// TIA Portal V20 export
FUNCTION_BLOCK "F-FB_DigitalOutput"   // FB111, F_LAD
{ S7_Optimized_Access := 'TRUE' }
// stored: AutoNumber false
BEGIN

REGION Network 1: Contactor for Machine
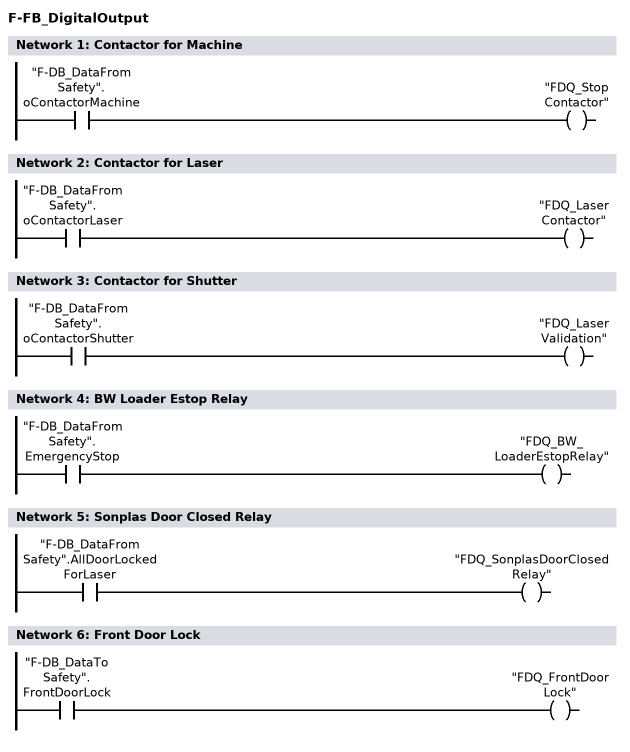
   RUNG wire#powerrail
      Contact( "F-DB_DataFromSafety".oContactorMachine )
      Coil( "FDQ_StopContactor" )
   END_RUNG
   // the same network as SCL:
   "FDQ_StopContactor" := "F-DB_DataFromSafety".oContactorMachine;
END_REGION

REGION Network 2: Contactor for Laser
   RUNG wire#powerrail
      Contact( "F-DB_DataFromSafety".oContactorLaser )
      Coil( "FDQ_LaserContactor" )
   END_RUNG
   // the same network as SCL:
   "FDQ_LaserContactor" := "F-DB_DataFromSafety".oContactorLaser;
END_REGION

REGION Network 3: Contactor for Shutter
   RUNG wire#powerrail
      Contact( "F-DB_DataFromSafety".oContactorShutter )
      Coil( "FDQ_LaserValidation" )
   END_RUNG
   // the same network as SCL:
   "FDQ_LaserValidation" := "F-DB_DataFromSafety".oContactorShutter;
END_REGION

REGION Network 4: BW Loader Estop Relay
   RUNG wire#powerrail
      Contact( "F-DB_DataFromSafety".EmergencyStop )
      Coil( "FDQ_BW_LoaderEstopRelay" )
   END_RUNG
   // the same network as SCL:
   "FDQ_BW_LoaderEstopRelay" := "F-DB_DataFromSafety".EmergencyStop;
END_REGION

REGION Network 5: Sonplas Door Closed Relay
   RUNG wire#powerrail
      Contact( "F-DB_DataFromSafety".AllDoorLockedForLaser )
      Coil( "FDQ_SonplasDoorClosedRelay" )
   END_RUNG
   // the same network as SCL:
   "FDQ_SonplasDoorClosedRelay" := "F-DB_DataFromSafety".AllDoorLockedForLaser;
END_REGION

REGION Network 6: Front Door Lock
   RUNG wire#powerrail
      Contact( "F-DB_DataToSafety".FrontDoorLock )
      Coil( "FDQ_FrontDoorLock" )
   END_RUNG
   // the same network as SCL:
   "FDQ_FrontDoorLock" := "F-DB_DataToSafety".FrontDoorLock;
END_REGION
END_FUNCTION_BLOCK
